// TIA Portal V19 export
FUNCTION "DEBUG_Simulate_Send_Msg_102" : Void   // FC215, LAD
TITLE = TEST INVIO MESSAGGIO 102
// stored: SetENOAutomatically false
   VAR_TEMP   // added for the SCL form of the ladder/FBD networks
      _w1 : Bool;
   END_VAR
BEGIN

REGION Network 1
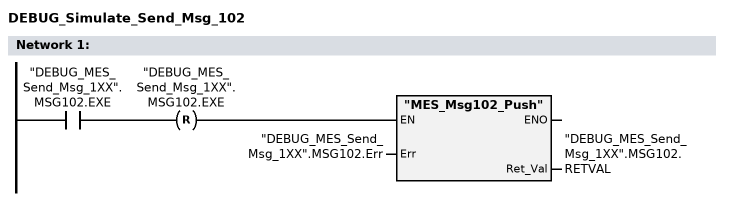
   RUNG wire#powerrail
      Contact( "DEBUG_MES_Send_Msg_1XX".MSG102.EXE )
      R_Coil( "DEBUG_MES_Send_Msg_1XX".MSG102.EXE )
      "MES_Msg102_Push"(Err := "DEBUG_MES_Send_Msg_1XX".MSG102.Err, Ret_Val => "DEBUG_MES_Send_Msg_1XX".MSG102.RETVAL)
   END_RUNG
   // the same network as SCL:
   #_w1 := "DEBUG_MES_Send_Msg_1XX".MSG102.EXE;
   IF #_w1 THEN
       "DEBUG_MES_Send_Msg_1XX".MSG102.EXE := FALSE;
       "DEBUG_MES_Send_Msg_1XX".MSG102.RETVAL := "MES_Msg102_Push"(Err := "DEBUG_MES_Send_Msg_1XX".MSG102.Err);
   END_IF;
END_REGION
END_FUNCTION
